PROGRAM ArmXYPosAdjust
VAR
	fbHMISimulateArmMovement_Arm1: fbHMISimulateArmMovement;
	fbHMISimulateArmMovement_Arm2: fbHMISimulateArmMovement;
	dummy2: LREAL;
	dummy1: LREAL;
END_VAR

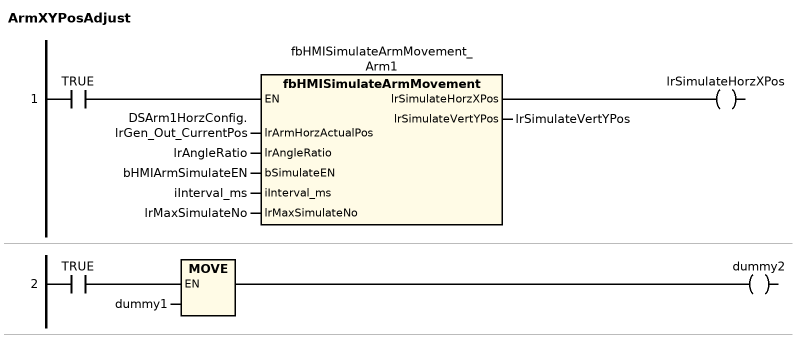
// NETWORK 1
fbHMISimulateArmMovement_Arm1(
    lrArmHorzActualPos := DSArm1HorzConfig.lrGen_Out_CurrentPos,
    lrAngleRatio := lrAngleRatio,
    bSimulateEN := bHMIArmSimulateEN,
    iInterval_ms := iInterval_ms,
    lrMaxSimulateNo := lrMaxSimulateNo,
    lrSimulateVertYPos => lrSimulateVertYPos); // fbHMISimulateArmMovement
lrSimulateHorzXPos := fbHMISimulateArmMovement_Arm1.lrSimulateHorzXPos;

// NETWORK 2
dummy2 := dummy1;

END_PROGRAM

(* stored: Version 1.1.0.1, ProductVersion 3.1.4024.12
   POU ArmXYPosAdjust: Id {2b985b6d-4aa4-408e-9e6b-a7221a54180d}, SpecialFunc None *)
